// TIA Portal V17 export
// export: Created 2025-01-16T19:22:27.65518Z, ExportSetting WithDefaults, DisplayName Totally Integrated Automation Portal, DisplayVersion V17 Update 6, DisplayName TIA Portal Openness, DisplayVersion V17 Update 6, DisplayName TIA Portal Version Control Interface, DisplayVersion V17, DisplayName STEP 7 Professional, DisplayVersion V17 Update 6, DisplayName STEP 7 Safety, DisplayVersion V17 Update 6, DisplayName WinCC Advanced, DisplayVersion V17 Update 6
VAR_GLOBAL   // PLC tag table "Default tag table"
   START AT %M0.0 : Bool;
   STOP AT %M0.1 : Bool;
   MOTOR AT %Q0.0 : Bool;
END_VAR
